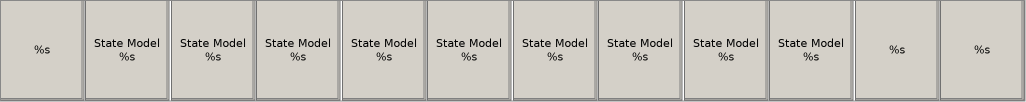
VISUALIZATION VIS_TemplateKeys  // 1026x102
VAR_INPUT
	Caption		: ARRAY [1..12] OF STRING;
END_VAR
VAR_IN_OUT
	KeyPressed	: ARRAY [1..12] OF BOOL;
END_VAR
    Button (0,0 84x100), "%s", text variable: Caption[1]
        tap KeyPressed[1]
    Button (85,0 84x100), "State Model %s", text variable: Caption[2]
        tap KeyPressed[2]
    Button (171,0 84x100), "State Model %s", text variable: Caption[3]
        tap KeyPressed[3]
    Button (256,0 84x100), "State Model %s", text variable: Caption[4]
        tap KeyPressed[4]
    Button (342,0 84x100), "State Model %s", text variable: Caption[5]
        tap KeyPressed[5]
    Button (427,0 84x100), "State Model %s", text variable: Caption[6]
        tap KeyPressed[6]
    Button (513,0 84x100), "State Model %s", text variable: Caption[7]
        tap KeyPressed[7]
    Button (598,0 84x100), "State Model %s", text variable: Caption[8]
        tap KeyPressed[8]
    Button (684,0 84x100), "State Model %s", text variable: Caption[9]
        tap KeyPressed[9]
    Button (769,0 84x100), "State Model %s", text variable: Caption[10]
        tap KeyPressed[10]
    Button (855,0 84x100), "%s", text variable: Caption[11]
        tap KeyPressed[11]
    Button (940,0 84x100), "%s", text variable: Caption[12]
        tap KeyPressed[12]
END_VISUALIZATION

(* stored: Version 1.1.0.1, ProductVersion 3.1.4024.12
   Visu VIS_TemplateKeys: Id {ff7448d5-17e6-41b2-8d2c-30a39d20dd9d} *)
